FUNCTION_BLOCK FB_TestBasic
VAR_INPUT
	DO0	: BOOL; // Enable the servo	
END_VAR
VAR_IN_OUT
	data	: ST_TestBasic;	// Ethernet IP data
END_VAR
VAR_OUTPUT
	DI0	: BOOL;
	Ready	: BOOL;
	Error	: UINT; 
END_VAR
VAR
END_VAR

METHOD OpcuaMonitor : BOOL
VAR_INPUT
END_VAR
VAR_IN_OUT
	Data	: ST_SpindleControl;
END_VAR
VAR_OUTPUT
	Error	: BOOL;
END_VAR
VAR_INST
	fbHbMonitor	: FB_HeartbeatMonitor;
END_VAR
fbHbMonitor(CLK:= Data.status.input.Heartbeat, PT:= T#2.5S, Q=> );

IF NOT fbHbMonitor.Q THEN
	MEMSET(ADR(Data.input), 0, SIZEOF(Data.input));
	Error := TRUE;
ELSE
	Error := FALSE;
END_IF
END_METHOD

END_FUNCTION_BLOCK

(* stored: Version 1.1.0.1, ProductVersion 3.1.4024.9
   POU FB_TestBasic: Id {ab1c2dc1-87be-467c-802a-8b1dc0728c8c}, SpecialFunc None
   Method OpcuaMonitor: Id {8a848c2d-bc78-4c2f-9235-a424d0e44822} *)
